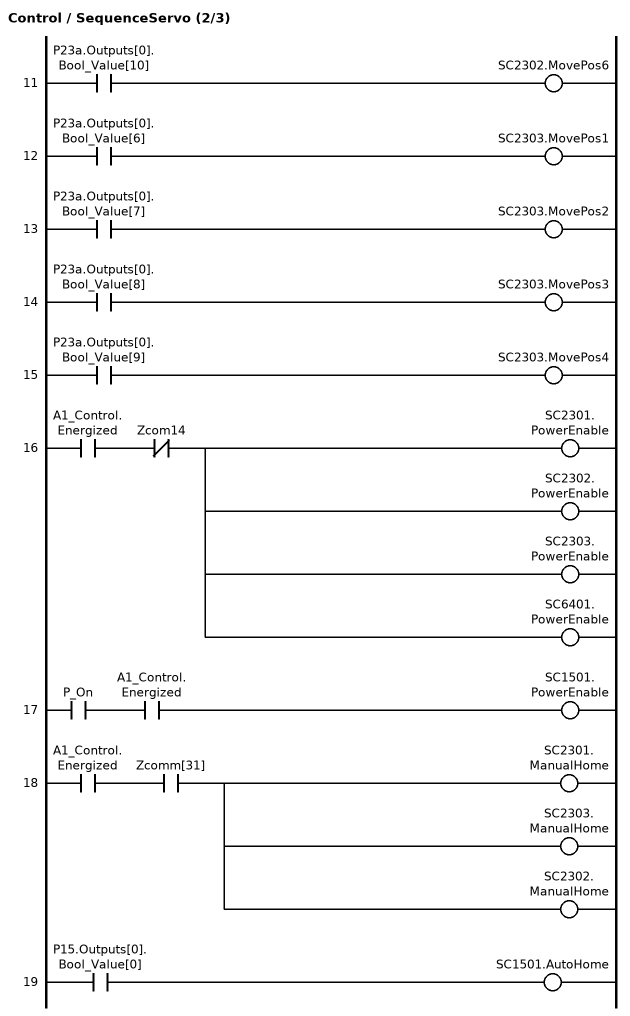
(* [picture p72: Control / SequenceServo, rungs 11-19] *)
(* Rung 11 *)
SC2302.MovePos6 := P23a.Outputs[0].Bool_Value[10];
(* Rung 12 *)
SC2303.MovePos1 := P23a.Outputs[0].Bool_Value[6];
(* Rung 13 *)
SC2303.MovePos2 := P23a.Outputs[0].Bool_Value[7];
(* Rung 14 *)
SC2303.MovePos3 := P23a.Outputs[0].Bool_Value[8];
(* Rung 15 *)
SC2303.MovePos4 := P23a.Outputs[0].Bool_Value[9];
(* Rung 16 *)
SC2301.PowerEnable := A1_Control.Energized AND NOT Zcom14;
SC2302.PowerEnable := A1_Control.Energized AND NOT Zcom14;
SC2303.PowerEnable := A1_Control.Energized AND NOT Zcom14;
SC6401.PowerEnable := A1_Control.Energized AND NOT Zcom14;
(* Rung 17 *)
SC1501.PowerEnable := P_On AND A1_Control.Energized;
(* Rung 18 *)
SC2301.ManualHome := A1_Control.Energized AND Zcomm[31];
SC2303.ManualHome := A1_Control.Energized AND Zcomm[31];
SC2302.ManualHome := A1_Control.Energized AND Zcomm[31];
(* Rung 19 *)
SC1501.AutoHome := P15.Outputs[0].Bool_Value[0];

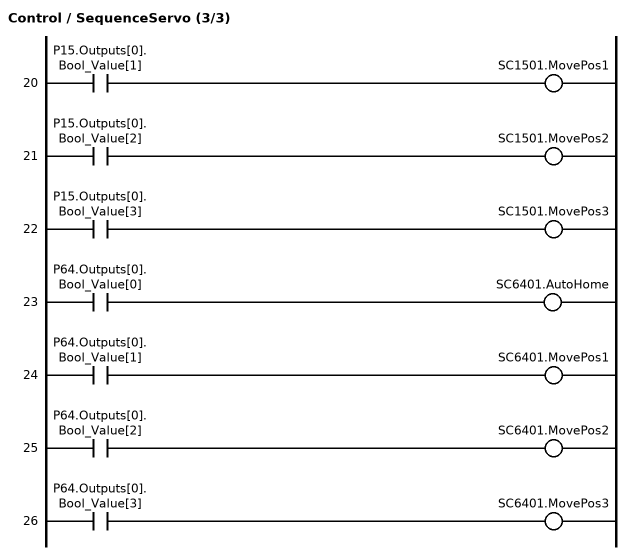
(* Rung 20 *)
SC1501.MovePos1 := P15.Outputs[0].Bool_Value[1];
(* Rung 21 *)
SC1501.MovePos2 := P15.Outputs[0].Bool_Value[2];
(* Rung 22 *)
SC1501.MovePos3 := P15.Outputs[0].Bool_Value[3];
(* Rung 23 *)
SC6401.AutoHome := P64.Outputs[0].Bool_Value[0];
(* Rung 24 *)
SC6401.MovePos1 := P64.Outputs[0].Bool_Value[1];
(* Rung 25 *)
SC6401.MovePos2 := P64.Outputs[0].Bool_Value[2];
(* Rung 26 *)
SC6401.MovePos3 := P64.Outputs[0].Bool_Value[3];

(* Section SequenceMotor: ladder, written here as Structured Text *)

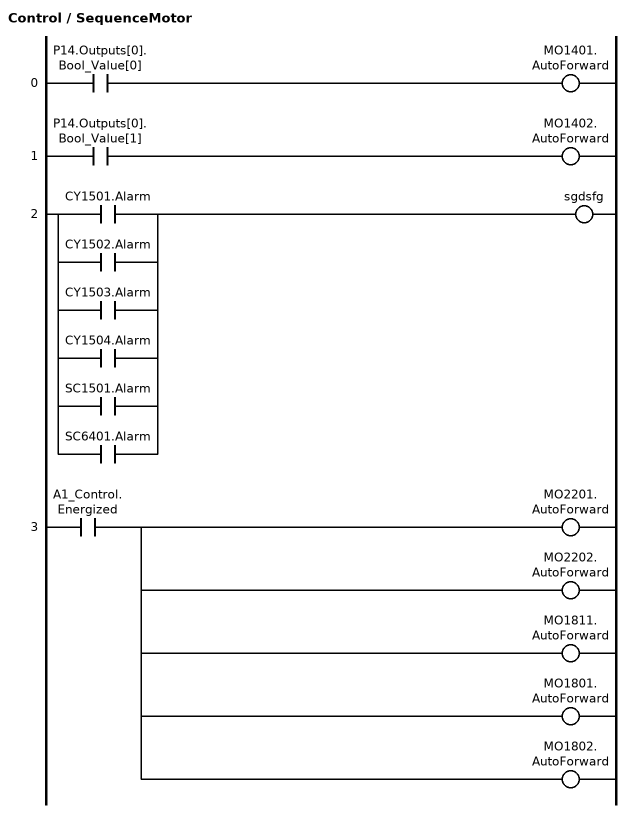
(* Rung 0 *)
MO1401.AutoForward := P14.Outputs[0].Bool_Value[0];
(* Rung 1 *)
MO1402.AutoForward := P14.Outputs[0].Bool_Value[1];
(* Rung 2 *)
sgdsfg := CY1501.Alarm OR CY1502.Alarm OR CY1503.Alarm OR CY1504.Alarm OR SC1501.Alarm OR SC6401.Alarm;
(* Rung 3 *)
MO2201.AutoForward := A1_Control.Energized;
MO2202.AutoForward := A1_Control.Energized;
MO1811.AutoForward := A1_Control.Energized;
MO1801.AutoForward := A1_Control.Energized;
MO1802.AutoForward := A1_Control.Energized;
END_PROGRAM

PROGRAM Outputs
VAR
    zcom : ARRAY[0..19] OF BOOL;
    IL0301_FB : MISCOUT;
    IL0302_FB : MISCOUT;
    IL0303_FB : MISCOUT;
    DO3501_FB : MISCOUT;
    DO1701_FB : MISCOUT;
    K1301_FB : MISCOUT;
    servo_drive_Error : BOOL;
    Actual_Value : DWORD;
    DO0351_FB : MISCOUT;
    CY1508_FB : CYL;
    CY1807_FB : CYL;
    CY1511_FB : CYL;
    CY1512_FB : CYL;
    CY3201_FB : CYL;
    CY3601_FB : CYL;
    SV1511_FB : MISCOUT;
    zcom1 : BOOL;
    zcom2 : BOOL;
    zcom6 : BOOL;
    CY4101_FB : CYL;
    CY4102_FB : CYL;
    CY4103_FB : CYL;
    CY4104_FB : CYL;
    CY4111_FB : CYL;
    CY4112_FB : CYL;
    CY4113_FB : CYL;
    CY4114_FB : CYL;
    CY4121_FB : CYL;
    CY4122_FB : CYL;
    CY4123_FB : CYL;
    CY4124_FB : CYL;
    Test2 : BOOL;
    SV : BOOL;
    SV4101_FB : MISCOUT;
    SV4102_FB : MISCOUT;
    SV4103_FB : MISCOUT;
    SV4104_FB : MISCOUT;
    XC0411_O1_15 : BOOL;
    MO1411_FB : MOTOR;
    zcom20 : BOOL;
    CY1401_FB : CYL;
    CY1402_FB : CYL;
    zcom21 : BOOL;
    zcom22 : BOOL;
    zcom23 : BOOL;
    zcom24 : BOOL;
    zcom_24 : BOOL;
    zcom_25 : BOOL;
    zcom_26 : BOOL;
    zcom_27 : BOOL;
    IL0304_FB : MiscOut;
    IL0305_FB : MiscOut;
    IL0306_FB : MiscOut;
    SV2701_FB : MiscOut;
    SV2702_FB : MiscOut;
    SV1501_FB : MiscOut;
    SV4111_FB : MiscOut;
    SV4112_FB : MiscOut;
    SV4113_FB : MiscOut;
    SV4114_FB : MiscOut;
    SV4121_FB : MiscOut;
    SV4122_FB : MiscOut;
    SV4123_FB : MiscOut;
    SV4124_FB : MiscOut;
    CY1501_FB : CYL;
    CY1502_FB : CYL;
    CY1503_FB : CYL;
    CY1504_FB : CYL;
    CY1505_FB : CYL;
    CY1506_FB : CYL;
    CY1507_FB : CYL;
    CY1801_FB : CYL;
    CY1802_FB : CYL;
    CY1804_FB : CYL;
    CY1803_FB : CYL;
    CY1805FB : CYL;
    CY1805_FB : CYL;
    CY1806_FB : CYL;
    CY2701_FB : CYL;
    CY3105_FB : CYL;
    SC1701_FB : Servo;
    SC2701_FB : Servo;
    SC_3201_FB : Servo;
    SC3201_FB : Servo;
    SC1702_FB : Servo;
    SC3601_FB : Servo;
    SC201_FB : Servo;
    SC3202_FB : Servo;
    MO2301_FB : Motor;
    MO3101_FB : MotorVSD;
    MO1401_FB : Motor;
    CY3102_FB : CYL;
    CY3103_FB : CYL;
    SC1701_Gear_SC1702 : MC_GearIn;
    A : BOOL;
    Vision_Test : Vision;
    Test4 : BOOL;
    Comm_DN : BOOL;
    SC1701_Gear_SC1702_Stop : MC_GearOut;
    GearStopMode : _eMC_OUT_MODE;
    CA2701_FB : Vision;
    CA1701_FB : Vision;
    SC1501_FB : Servo;
    CY1513_FB : CYL;
    CY1514_FB : CYL;
    CY1514_Extend : BOOL;
    CY1514_Retract : BOOL;
    CY3101_FB : CYL;
    SV4105_FB : MiscOut;
    SV4106_FB : MiscOut;
    SV4107_FB : MiscOut;
    SV4108_FB : MiscOut;
    SV4115_FB : MiscOut;
    SV4116_FB : MiscOut;
    SV4117_FB : MiscOut;
    SV4118_FB : MiscOut;
    SV4125_FB : MiscOut;
    SV4126_FB : MiscOut;
    SV4127_FB : MiscOut;
    SV4128_FB : MiscOut;
    CY1601_FB : CYL;
    CY1602_FB : CYL;
    CY2201_FB : CYL;
    CY2301_FB : CYL;
    CY2302_FB : CYL;
    CY2303_FB : CYL;
    CY2311_FB : CYL;
    CY2312_FB : CYL;
    CY2313_FB : CYL;
    CY2314_FB : CYL;
    CY2315_FB : CYL;
    CY2316_FB : CYL;
    CY2317_FB : CYL;
    CY2318_FB : CYL;
    CY2319_FB : CYL;
    CY2401_FB : CYL;
    CY2402_FB : CYL;
    MO1402_FB : Motor;
    MO3401_FB : MotorVSD;
    MO2311_FB : Motor;
    MO2201_FB : Motor;
    MO2202_FB : Motor;
    CY2501_A_FB : CYL;
    CY2501_B_FB : CYL;
    CY2501_C_FB : CYL;
    CY2501_D_FB : CYL;
    CY2502_A_FB : CYL;
    CY2502_B_FB : CYL;
    CY2503_A_FB : CYL;
    CY2503_B_FB : CYL;
    DO0301_FB : MiscOut;
    K0320_FB : MiscOut;
    K0321_FB : MiscOut;
    K0322_FB : MiscOut;
    K0323_FB : MiscOut;
    K4001_FB : MiscOut;
    DO3301_FB : MiscOut;
    DO3302_FB : MiscOut;
    SV0401_FB : MiscOut;
    SV2301_FB : MiscOut;
    SV2311_FB : MiscOut;
    SV2501_FB : MiscOut;
    SV2502_FB : MiscOut;
    CY3101_B_FB : CYL;
    CY3104_FB : CYL;
    CY3106_FB : CYL;
    CY2304_FB : CYL;
    CY2305_FB : CYL;
    CY2306_FB : CYL;
    CY2307_FB : CYL;
    CY2308_FB : CYL;
    CY2309_FB : CYL;
    M03401_FB : Motor;
    c : DINT;
    CY2501_FB : CYL;
    CY2502_FB : CYL;
    xc : BOOL;
    CY2201EX : BOOL;
    CY2201RT : BOOL;
    DO3502_FB : MiscOut;
    SV1502_FB : MiscOut;
    SV1503_FB : MiscOut;
    SV2511_FB : MiscOut;
    SV2512_FB : MiscOut;
    SV2521_FB : MiscOut;
    SV7101_FB : MiscOut;
    DO0320_FB : MiscOut;
    DO0350_FB : MiscOut;
    CY1811_FB : CYL;
    CY1812_FB : CYL;
    CY1701_FB : CYL;
    CY1702_FB : CYL;
    CY1703_FB : CYL;
    CY2521_FB : CYL;
    CY7101_FB : CYL;
    CY7102_FB : CYL;
    CY3401_FB : CYL;
    MO1801_FB : Motor;
    MO1811_FB : Motor;
    MO1701_FB : Motor;
    SC6401_FB : Servo;
    SC2301_FB : Servo;
    SC2302_FB : Servo;
    SC2303_FB : Servo;
    DO3511_FB : MiscOut;
    CY3402_FB : CYL;
    M03101_FB : Motor;
    MO2701_FB : Motor;
    MO2702_FB : Motor;
    MO1802_FB : Motor;
    SV2522_FB : MiscOut;
END_VAR
VAR_EXTERNAL
    CY1601 : CylinderD;
    A1_Control : System;
    CY2502 : CylinderD;
    CY2501 : CylinderD;
    CY2402 : CylinderD;
    CY2401 : CylinderD;
    CY2302 : CylinderD;
    CY2303 : CylinderD;
    CY2301 : CylinderD;
    SC2701 : ServoD;
    MO1402 : MotorD;
    MO2301 : MotorD;
    MO2201 : MotorD;
    MO2202 : MotorD;
    IL0302 : MiscOutD;
    IL0303 : MiscOutD;
    DO0301 : MiscOutD;
    DO3301 : MiscOutD;
    DO3302 : MiscOutD;
    SV0401 : MiscOutD;
    SV1501 : MiscOutD;
    SV2301 : MiscOutD;
    SV2501 : MiscOutD;
    SV2502 : MiscOutD;
    IL0301 : MiscOutD;
    CY2304 : CylinderD;
    RO4001_I_PalletizingDone : BOOL;
    PS2501 : MiscInD;
    P27 : SequenceD;
    SKU_Select : DINT;
    DO3502 : MiscOutD;
    DO3501 : MiscOutD;
    K1301 : MiscOutD;
    SV2701 : MiscOutD;
    SV1502 : MiscOutD;
    SV1503 : MiscOutD;
    SV2511 : MiscOutD;
    SV2512 : MiscOutD;
    SV2521 : MiscOutD;
    SV7101 : MiscOutD;
    DO320 : MiscOutD;
    DO0320 : MiscOutD;
    DO0350 : MiscOutD;
    CY1502 : CylinderD;
    CY1503 : CylinderD;
    CY1504 : CylinderD;
    CY1811 : CylinderD;
    CY1701 : CylinderD;
    CY1702 : CylinderD;
    CY1703 : CylinderD;
    CY2521 : CylinderD;
    CY7101 : CylinderD;
    CY7102 : CylinderD;
    CY3401 : CylinderD;
    CY3402 : CylinderD;
    MO1801 : MotorD;
    MO1811 : MotorD;
    MO1701 : MotorD;
    MO3101 : MotorD;
    SC1501 : ServoD;
    SC1501_Ax : _sAXIS_REF;
    SC6401 : ServoD;
    SC6401_Ax : _sAXIS_REF;
    SC2301 : ServoD;
    SC2301_Ax : _sAXIS_REF;
    SC2302 : ServoD;
    SC2302_Ax : _sAXIS_REF;
    SC2303 : ServoD;
    SC2303_Ax : _sAXIS_REF;
    XC0301_6_I : ARRAY[0..15] OF BOOL;
    XC0301_7_I : ARRAY[0..15] OF BOOL;
    XC0301_8_O : ARRAY[0..15] OF BOol;
    IL0304 : MiscOutD;
    XC0301_9_O : ARRAY[0..15] OF BOOL;
    XC0320_1_O_2 : BOOL;
    XC0320_1_O_3 : BOOL;
    XC0320_1_O_4 : BOOL;
    XC0320_1_I_5 : BOOL;
    XC0320_1_I_6 : BOOL;
    XC0320_1_I_7 : BOOL;
    XC0320_1_I_8 : BOOL;
    XC0320_1_I_9 : BOOL;
    XC0320_1_I_10 : BOOL;
    XC0320_2_O_0 : BOOL;
    XC0320_2_O_1 : BOOL;
    XC0320_2_O_2 : BOOL;
    XC0320_2_O_3 : BOOL;
    XC0320_2_O_4 : BOOL;
    XC0320_2_O_5 : BOOL;
    DO3511 : MiscOutD;
    XC0320_2_O_6 : BOOL;
    XC0320_3_O_0 : BOOL;
    XC0320_3_O_1 : BOOL;
    XC0320_3_O_2 : BOOL;
    XC0320_3_O_3 : BOOL;
    XC0320_3_I_4 : BOOL;
    XC0320_3_I_5 : BOOL;
    XC0320_3_I_6 : BOOL;
    XC0320_3_I_7 : BOOL;
    XC0320_3_I_8 : BOOL;
    XC0320_3_I_9 : BOOL;
    XC0320_4_I_0 : BOOL;
    XC0320_4_I_1 : BOOL;
    XC0320_4_I_2 : BOOL;
    XC0320_4_I_3 : BOOL;
    XC0320_4_I_4 : BOOL;
    XC0320_4_I_5 : BOOL;
    XC0320_4_I_6 : BOOL;
    XC0320_4_I_7 : BOOL;
    XC0320_4_I_8 : BOOL;
    XC0320_4_I_9 : BOOL;
    XC0320_4_I_10 : BOOL;
    XC0320_4_I_11 : BOOL;
    XC0320_4_I_12 : BOOL;
    XC0320_4_I_13 : BOOL;
    XC0320_4_I_14 : BOOL;
    XC0320_4_I_15 : BOOL;
    XC0320_5_I_0 : BOOL;
    XC0320_5_I_1 : BOOL;
    XC0320_5_I_2 : BOOL;
    XC0320_5_I_3 : BOOL;
    MO1401 : MotorD;
    MO3401 : MotorD;
    CY1501 : CylinderD;
    Ketan : WORD;
    Sandesh : WORD;
    jhsac : BOOL;
    CY2305 : CylinderD;
    XC0320_1_I_0 : BOOL;
    XC0320_1_I_1 : BOOL;
    XC0320_1_I_11 : BOOL;
    XC0320_1_I_12 : BOOL;
    XC0320_3_I_14 : BOOL;
    XC0320_3_I_15 : BOOL;
    XC0320_5_O_8 : BOOL;
    XC0320_5_O_9 : BOOL;
    XC0320_5_O_10 : BOOL;
    MO2701 : MotorD;
    MO2702 : MotorD;
    MO1802 : MotorD;
    SV2522 : MiscOutD;
    A0XC0401_1_I_4 : BOOL;
    A0XC0401_1_I_5 : BOOL;
    A0XC0401_1_I_6 : BOOL;
    A0XC0401_1_I_7 : BOOL;
    CY2701 : CylinderD;
    A0XC0401_1_I_11 : BOOL;
    A0XC0401_1_I_12 : BOOL;
    A0XC0401_1_O_0 : BOOL;
    A0XC0401_1_O_1 : BOOL;
    A0XC0401_1_O_3 : BOOL;
    A0XC0401_1_O_4 : BOOL;
    A0XC0401_1_O_5 : BOOL;
    A0XC0401_1_O_2 : BOOL;
    A0XC0401_2_O_0 : BOOL;
    A0XC0401_2_O_1 : BOOL;
    A0XC0401_1_O_6 : BOOL;
    A0XC0401_1_O_7 : BOOL;
    XC0320_1_I_15 : BOOL;
    XC0320_1_I_14 : BOOL;
    A0XC0401_2_O_2 : BOOL;
    A0XC0401_2_O_3 : BOOL;
    A0XC0401_2_O_4 : BOOL;
    A0XC0401_2_O_5 : BOOL;
    A0XC0401_2_O_6 : BOOL;
    A0XC0401_2_O_7 : BOOL;
END_VAR
VAR_EXTERNAL CONSTANT
    SC1501Ax : _sAXIS_REF;
    SC2301Ax : _sAXIS_REF;
    SC2302Ax : _sAXIS_REF;
    SC2303Ax : _sAXIS_REF;
    SC6401Ax : _sAXIS_REF;
END_VAR
VAR_EXTERNAL
    XC0320_2_O_8 : BOOL;
    XC0320_2_O_9 : BOOL;
    A0XC0401_3_O_0 : BOOL;
    A0XC0401_3_O_1 : BOOL;
    A0XC0401_3_O_2 : BOOL;
    A0XC0401_3_O_3 : BOOL;
    A0XC0401_3_O_4 : BOOL;
    A0XC0401_3_O_5 : BOOL;
    A0XC0401_3_O_6 : BOOL;
    A0XC0401_3_O_7 : BOOL;
    XC0320_2_I_0 : BOOL;
    XC0320_2_I_1 : BOOL;
END_VAR

(* Section IDMiscOut: ladder, written here as Structured Text *)

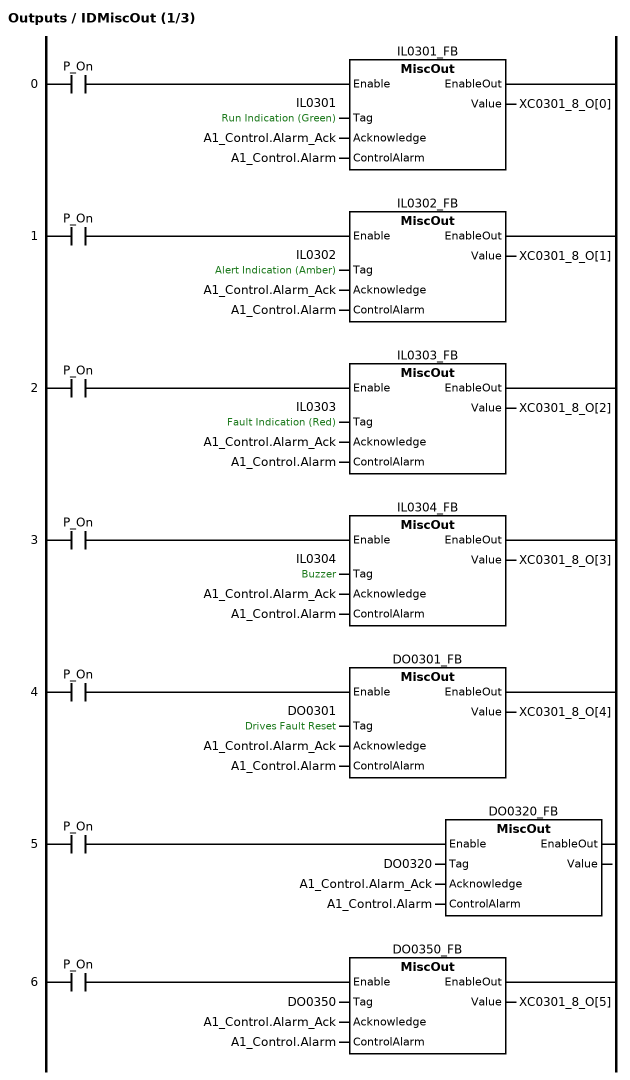
(* Rung 0 *)
IL0301_FB(Enable := P_On, Tag := IL0301, Acknowledge := A1_Control.Alarm_Ack, ControlAlarm := A1_Control.Alarm, Value => XC0301_8_O[0]);
(* Rung 1 *)
IL0302_FB(Enable := P_On, Tag := IL0302, Acknowledge := A1_Control.Alarm_Ack, ControlAlarm := A1_Control.Alarm, Value => XC0301_8_O[1]);
(* Rung 2 *)
IL0303_FB(Enable := P_On, Tag := IL0303, Acknowledge := A1_Control.Alarm_Ack, ControlAlarm := A1_Control.Alarm, Value => XC0301_8_O[2]);
(* Rung 3 *)
IL0304_FB(Enable := P_On, Tag := IL0304, Acknowledge := A1_Control.Alarm_Ack, ControlAlarm := A1_Control.Alarm, Value => XC0301_8_O[3]);
(* Rung 4 *)
DO0301_FB(Enable := P_On, Tag := DO0301, Acknowledge := A1_Control.Alarm_Ack, ControlAlarm := A1_Control.Alarm, Value => XC0301_8_O[4]);
(* Rung 5 *)
DO0320_FB(Enable := P_On, Tag := DO0320, Acknowledge := A1_Control.Alarm_Ack, ControlAlarm := A1_Control.Alarm);
(* notes on elements: Safety Reset *)
(* Rung 6 *)
DO0350_FB(Enable := P_On, Tag := DO0350, Acknowledge := A1_Control.Alarm_Ack, ControlAlarm := A1_Control.Alarm, Value => XC0301_8_O[5]);
(* notes on elements: Upstream Signal *)

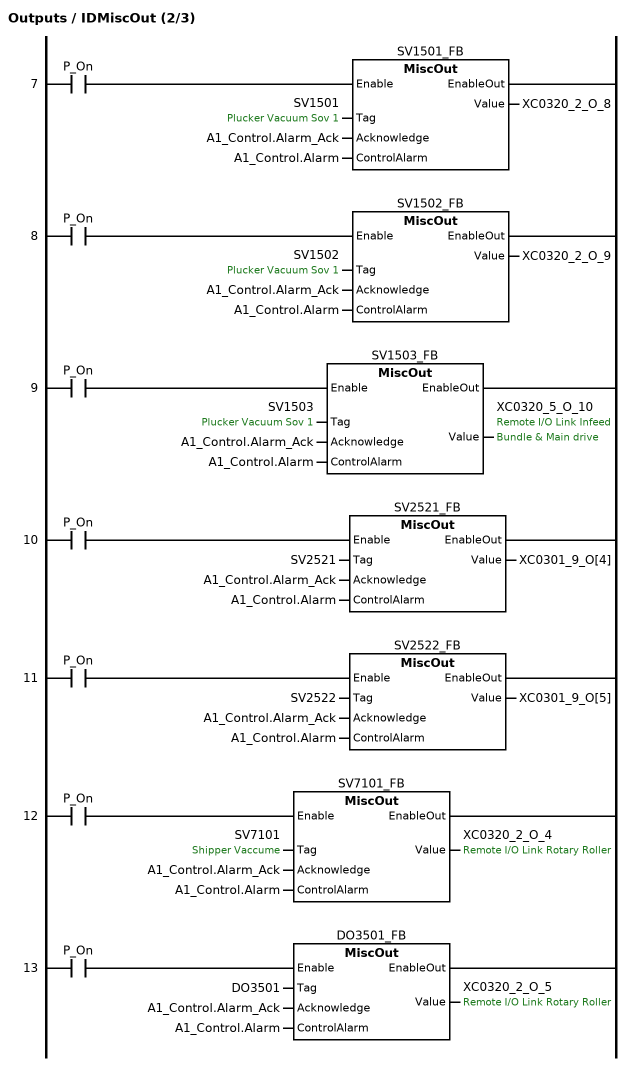
(* Rung 7 *)
SV1501_FB(Enable := P_On, Tag := SV1501, Acknowledge := A1_Control.Alarm_Ack, ControlAlarm := A1_Control.Alarm, Value => XC0320_2_O_8);
(* notes on elements: Plucker Vacuum Sov 1 *)
(* Rung 8 *)
SV1502_FB(Enable := P_On, Tag := SV1502, Acknowledge := A1_Control.Alarm_Ack, ControlAlarm := A1_Control.Alarm, Value => XC0320_2_O_9);
(* notes on elements: Plucker Vacuum Sov 2 *)
(* Rung 9 *)
SV1503_FB(Enable := P_On, Tag := SV1503, Acknowledge := A1_Control.Alarm_Ack, ControlAlarm := A1_Control.Alarm, Value => XC0320_5_O_10);
(* notes on elements: Plucker Vacuum Sov 3 *)
(* Rung 10 *)
SV2521_FB(Enable := P_On, Tag := SV2521, Acknowledge := A1_Control.Alarm_Ack, ControlAlarm := A1_Control.Alarm, Value => XC0301_9_O[4]);
(* notes on elements: Vacuum Solenoid *)
(* Rung 11 *)
SV2522_FB(Enable := P_On, Tag := SV2522, Acknowledge := A1_Control.Alarm_Ack, ControlAlarm := A1_Control.Alarm, Value => XC0301_9_O[5]);
(* notes on elements: layerboard pickhead purging *)
(* Rung 12 *)
SV7101_FB(Enable := P_On, Tag := SV7101, Acknowledge := A1_Control.Alarm_Ack, ControlAlarm := A1_Control.Alarm, Value => XC0320_2_O_4);
(* notes on elements: Shipper Vacuum *)
(* Rung 13 *)
DO3501_FB(Enable := P_On, Tag := DO3501, Acknowledge := A1_Control.Alarm_Ack, ControlAlarm := A1_Control.Alarm, Value => XC0320_2_O_5);
(* notes on elements: Pre-Label Applicator Trigger Signal *)

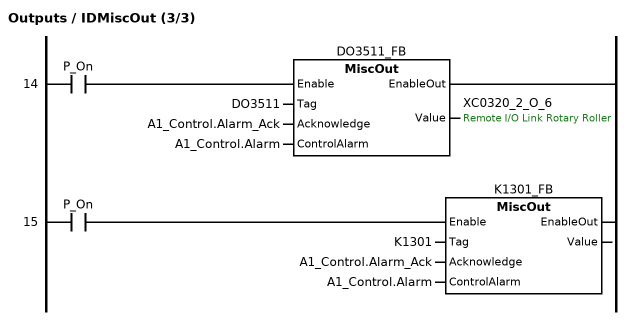
(* Rung 14 *)
DO3511_FB(Enable := P_On, Tag := DO3511, Acknowledge := A1_Control.Alarm_Ack, ControlAlarm := A1_Control.Alarm, Value => XC0320_2_O_6);
(* notes on elements: OCR Camera Trigger Signal *)
(* Rung 15 *)
K1301_FB(Enable := P_On, Tag := K1301, Acknowledge := A1_Control.Alarm_Ack, ControlAlarm := A1_Control.Alarm);
(* notes on elements: Guard Door Coil Supply *)

(* Section IDCylinder: ladder, written here as Structured Text *)

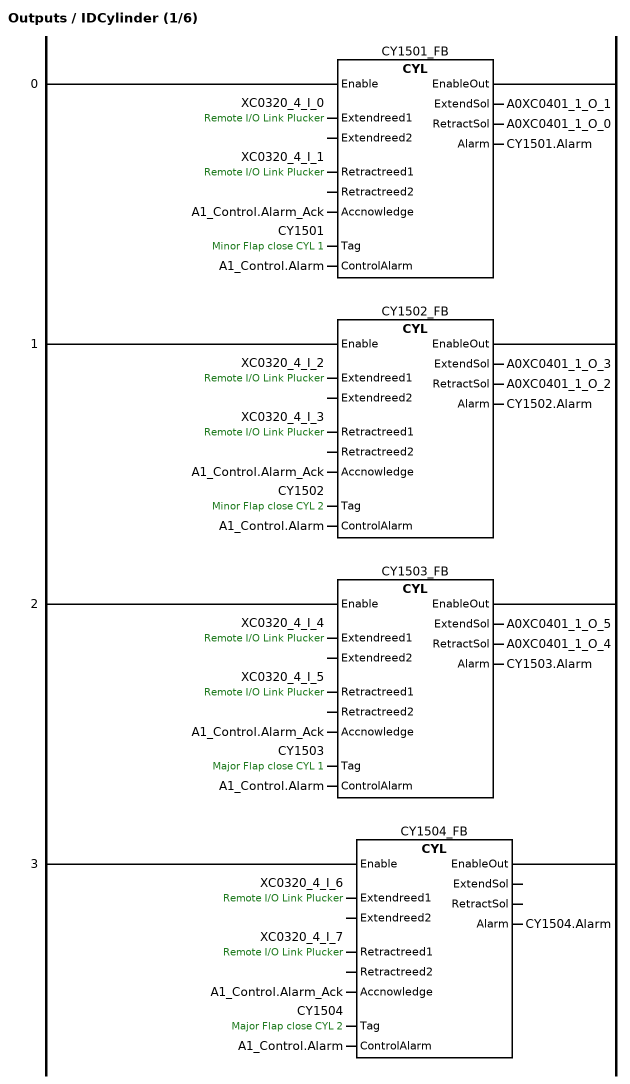
(* Rung 0 *)
CY1501_FB(Enable := TRUE, Extendreed1 := XC0320_4_I_0, Retractreed1 := XC0320_4_I_1, Accnowledge := A1_Control.Alarm_Ack, Tag := CY1501, ControlAlarm := A1_Control.Alarm, ExtendSol => A0XC0401_1_O_1, RetractSol => A0XC0401_1_O_0, Alarm => CY1501.Alarm);
(* notes on elements: Minor Flap close CYL 1 *)
(* Rung 1 *)
CY1502_FB(Enable := TRUE, Extendreed1 := XC0320_4_I_2, Retractreed1 := XC0320_4_I_3, Accnowledge := A1_Control.Alarm_Ack, Tag := CY1502, ControlAlarm := A1_Control.Alarm, ExtendSol => A0XC0401_1_O_3, RetractSol => A0XC0401_1_O_2, Alarm => CY1502.Alarm);
(* notes on elements: Minor Flap close CYL 2 *)
(* Rung 2 *)
CY1503_FB(Enable := TRUE, Extendreed1 := XC0320_4_I_4, Retractreed1 := XC0320_4_I_5, Accnowledge := A1_Control.Alarm_Ack, Tag := CY1503, ControlAlarm := A1_Control.Alarm, ExtendSol => A0XC0401_1_O_5, RetractSol => A0XC0401_1_O_4, Alarm => CY1503.Alarm);
(* notes on elements: Major Flap close CYL 1 *)
(* Rung 3 *)
CY1504_FB(Enable := TRUE, Extendreed1 := XC0320_4_I_6, Retractreed1 := XC0320_4_I_7, Accnowledge := A1_Control.Alarm_Ack, Tag := CY1504, ControlAlarm := A1_Control.Alarm, Alarm => CY1504.Alarm);
(* notes on elements: Major Flap close CYL 2 *)

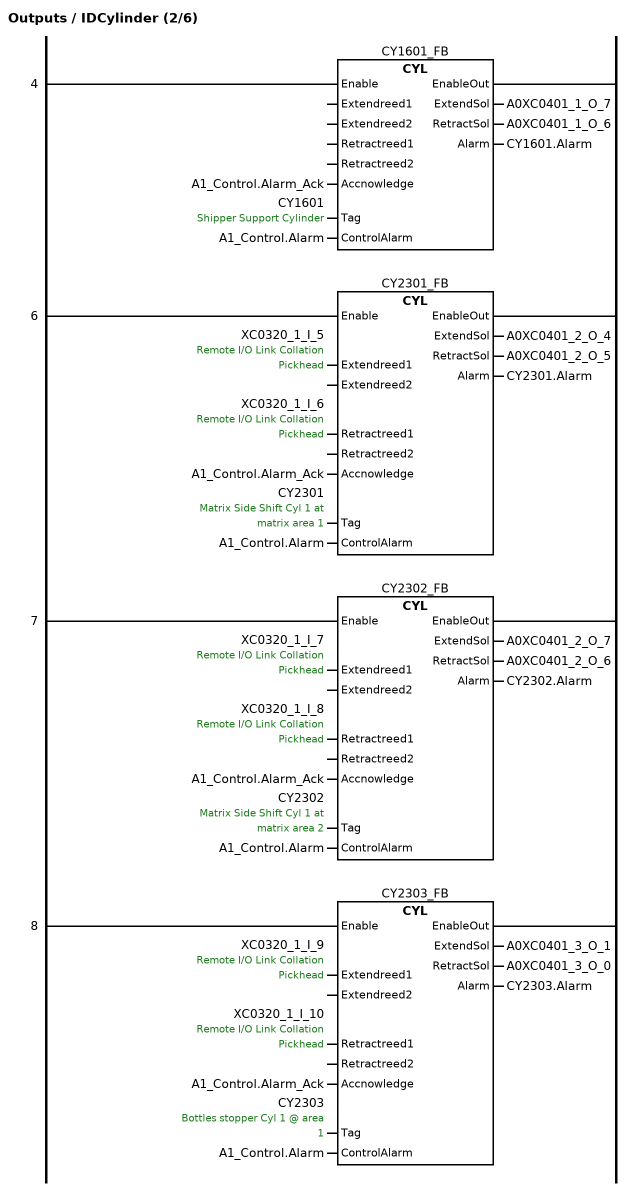
(* Rung 4 *)
CY1601_FB(Enable := TRUE, Accnowledge := A1_Control.Alarm_Ack, Tag := CY1601, ControlAlarm := A1_Control.Alarm, ExtendSol => A0XC0401_1_O_7, RetractSol => A0XC0401_1_O_6, Alarm => CY1601.Alarm);
(* Rung 6 *)
CY2301_FB(Enable := TRUE, Extendreed1 := XC0320_1_I_5, Retractreed1 := XC0320_1_I_6, Accnowledge := A1_Control.Alarm_Ack, Tag := CY2301, ControlAlarm := A1_Control.Alarm, ExtendSol => A0XC0401_2_O_4, RetractSol => A0XC0401_2_O_5, Alarm => CY2301.Alarm);
(* notes on elements: Matrix Side Shift Cyl 1 at matrix area 1 *)
(* Rung 7 *)
CY2302_FB(Enable := TRUE, Extendreed1 := XC0320_1_I_7, Retractreed1 := XC0320_1_I_8, Accnowledge := A1_Control.Alarm_Ack, Tag := CY2302, ControlAlarm := A1_Control.Alarm, ExtendSol => A0XC0401_2_O_7, RetractSol => A0XC0401_2_O_6, Alarm => CY2302.Alarm);
(* notes on elements: Matrix Side Shift Cyl 2 at matrix area 2 *)
(* Rung 8 *)
CY2303_FB(Enable := TRUE, Extendreed1 := XC0320_1_I_9, Retractreed1 := XC0320_1_I_10, Accnowledge := A1_Control.Alarm_Ack, Tag := CY2303, ControlAlarm := A1_Control.Alarm, ExtendSol => A0XC0401_3_O_1, RetractSol => A0XC0401_3_O_0, Alarm => CY2303.Alarm);

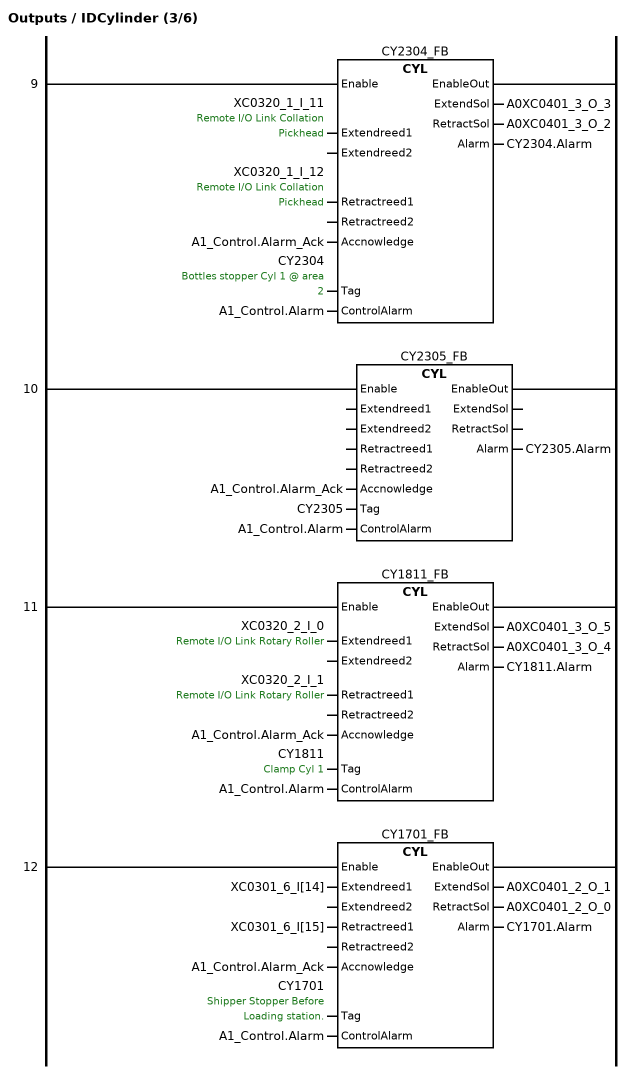
(* Rung 9 *)
CY2304_FB(Enable := TRUE, Extendreed1 := XC0320_1_I_11, Retractreed1 := XC0320_1_I_12, Accnowledge := A1_Control.Alarm_Ack, Tag := CY2304, ControlAlarm := A1_Control.Alarm, ExtendSol => A0XC0401_3_O_3, RetractSol => A0XC0401_3_O_2, Alarm => CY2304.Alarm);
(* notes on elements: Bottles stopper Cyl 1 @ area 1 *)
(* Rung 10 *)
CY2305_FB(Enable := TRUE, Accnowledge := A1_Control.Alarm_Ack, Tag := CY2305, ControlAlarm := A1_Control.Alarm, Alarm => CY2305.Alarm);
(* notes on elements: Bottles stopper Cyl 2 @ area 2 *)
(* Rung 11 *)
CY1811_FB(Enable := TRUE, Extendreed1 := XC0320_2_I_0, Retractreed1 := XC0320_2_I_1, Accnowledge := A1_Control.Alarm_Ack, Tag := CY1811, ControlAlarm := A1_Control.Alarm, ExtendSol => A0XC0401_3_O_5, RetractSol => A0XC0401_3_O_4, Alarm => CY1811.Alarm);
(* notes on elements: Clamp Cyl 1 *)
(* Rung 12 *)
CY1701_FB(Enable := TRUE, Extendreed1 := XC0301_6_I[14], Retractreed1 := XC0301_6_I[15], Accnowledge := A1_Control.Alarm_Ack, Tag := CY1701, ControlAlarm := A1_Control.Alarm, ExtendSol => A0XC0401_2_O_1, RetractSol => A0XC0401_2_O_0, Alarm => CY1701.Alarm);
(* notes on elements: Shipper Stopper Before Loading station. *)

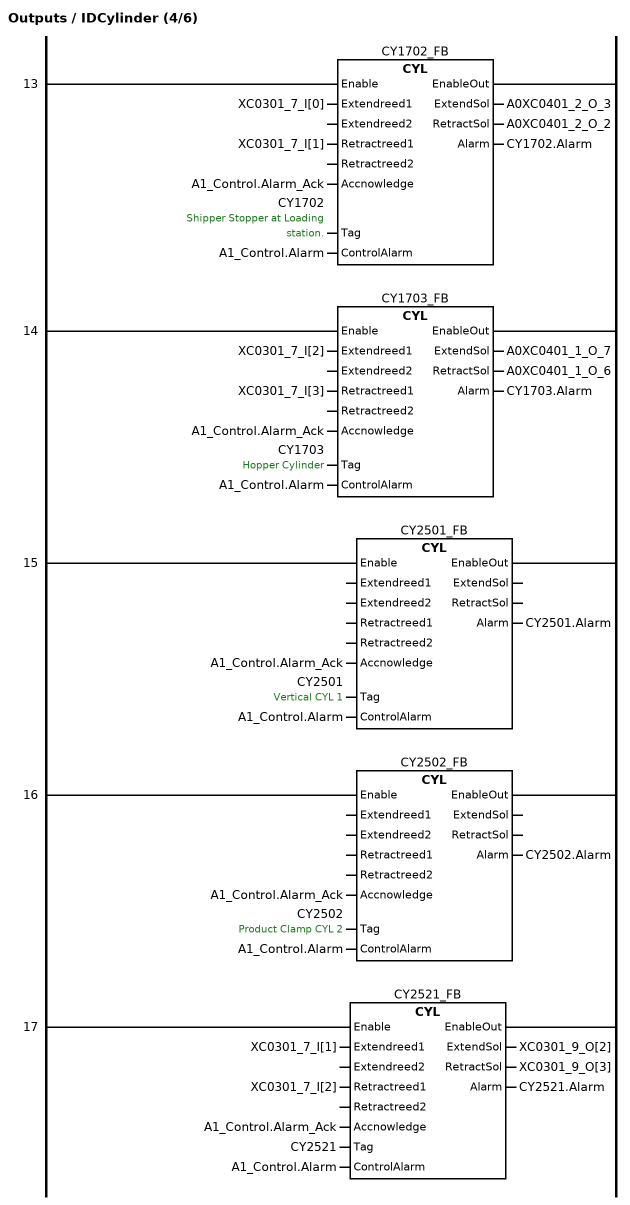
(* Rung 13 *)
CY1702_FB(Enable := TRUE, Extendreed1 := XC0301_7_I[0], Retractreed1 := XC0301_7_I[1], Accnowledge := A1_Control.Alarm_Ack, Tag := CY1702, ControlAlarm := A1_Control.Alarm, ExtendSol => A0XC0401_2_O_3, RetractSol => A0XC0401_2_O_2, Alarm => CY1702.Alarm);
(* notes on elements: Shipper Stopper at Loading station. *)
(* Rung 14 *)
CY1703_FB(Enable := TRUE, Extendreed1 := XC0301_7_I[2], Retractreed1 := XC0301_7_I[3], Accnowledge := A1_Control.Alarm_Ack, Tag := CY1703, ControlAlarm := A1_Control.Alarm, ExtendSol => A0XC0401_1_O_7, RetractSol => A0XC0401_1_O_6, Alarm => CY1703.Alarm);
(* notes on elements: Hopper Flap Open CYL *)
(* Rung 15 *)
CY2501_FB(Enable := TRUE, Accnowledge := A1_Control.Alarm_Ack, Tag := CY2501, ControlAlarm := A1_Control.Alarm, Alarm => CY2501.Alarm);
(* notes on elements: Bottle Clamp Cyl 1 *)
(* Rung 16 *)
CY2502_FB(Enable := TRUE, Accnowledge := A1_Control.Alarm_Ack, Tag := CY2502, ControlAlarm := A1_Control.Alarm, Alarm => CY2502.Alarm);
(* notes on elements: Bundle matrix clamp Cyl 1 *)
(* Rung 17 *)
CY2521_FB(Enable := TRUE, Extendreed1 := XC0301_7_I[1], Retractreed1 := XC0301_7_I[2], Accnowledge := A1_Control.Alarm_Ack, Tag := CY2521, ControlAlarm := A1_Control.Alarm, ExtendSol => XC0301_9_O[2], RetractSol => XC0301_9_O[3], Alarm => CY2521.Alarm);
(* notes on elements: Pickhead Rotary CYL *)

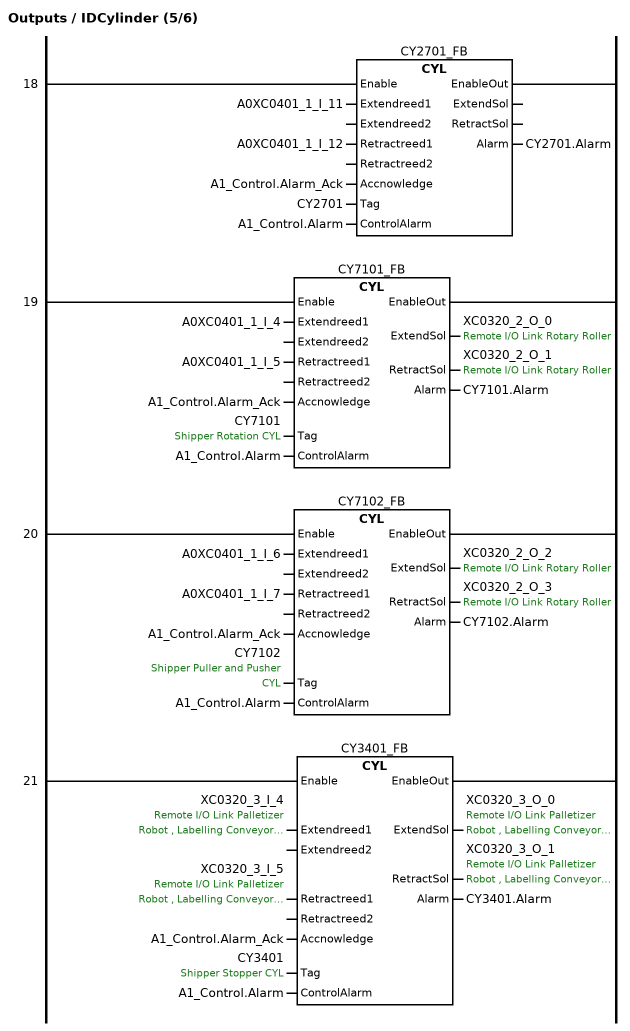
(* Rung 18 *)
CY2701_FB(Enable := TRUE, Extendreed1 := A0XC0401_1_I_11, Retractreed1 := A0XC0401_1_I_12, Accnowledge := A1_Control.Alarm_Ack, Tag := CY2701, ControlAlarm := A1_Control.Alarm, Alarm => CY2701.Alarm);
(* notes on elements: Minor Flap Close CYL @ Top Tapping *)
(* Rung 19 *)
CY7101_FB(Enable := TRUE, Extendreed1 := A0XC0401_1_I_4, Retractreed1 := A0XC0401_1_I_5, Accnowledge := A1_Control.Alarm_Ack, Tag := CY7101, ControlAlarm := A1_Control.Alarm, ExtendSol => XC0320_2_O_0, RetractSol => XC0320_2_O_1, Alarm => CY7101.Alarm);
(* notes on elements: Shipper Rotation CYL *)
(* Rung 20 *)
CY7102_FB(Enable := TRUE, Extendreed1 := A0XC0401_1_I_6, Retractreed1 := A0XC0401_1_I_7, Accnowledge := A1_Control.Alarm_Ack, Tag := CY7102, ControlAlarm := A1_Control.Alarm, ExtendSol => XC0320_2_O_2, RetractSol => XC0320_2_O_3, Alarm => CY7102.Alarm);
(* notes on elements: Shipper Puller and Pusher CYL *)
(* Rung 21 *)
CY3401_FB(Enable := TRUE, Extendreed1 := XC0320_3_I_4, Retractreed1 := XC0320_3_I_5, Accnowledge := A1_Control.Alarm_Ack, Tag := CY3401, ControlAlarm := A1_Control.Alarm, ExtendSol => XC0320_3_O_0, RetractSol => XC0320_3_O_1, Alarm => CY3401.Alarm);
(* notes on elements: Shipper Stopper Cylinder *)

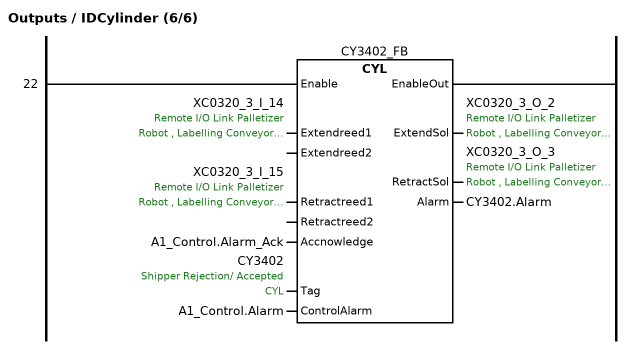
(* Rung 22 *)
CY3402_FB(Enable := TRUE, Extendreed1 := XC0320_3_I_14, Retractreed1 := XC0320_3_I_15, Accnowledge := A1_Control.Alarm_Ack, Tag := CY3402, ControlAlarm := A1_Control.Alarm, ExtendSol => XC0320_3_O_2, RetractSol => XC0320_3_O_3, Alarm => CY3402.Alarm);
(* notes on elements: Shipper Rejection CYL *)

(* Section IDServo: ladder, written here as Structured Text *)

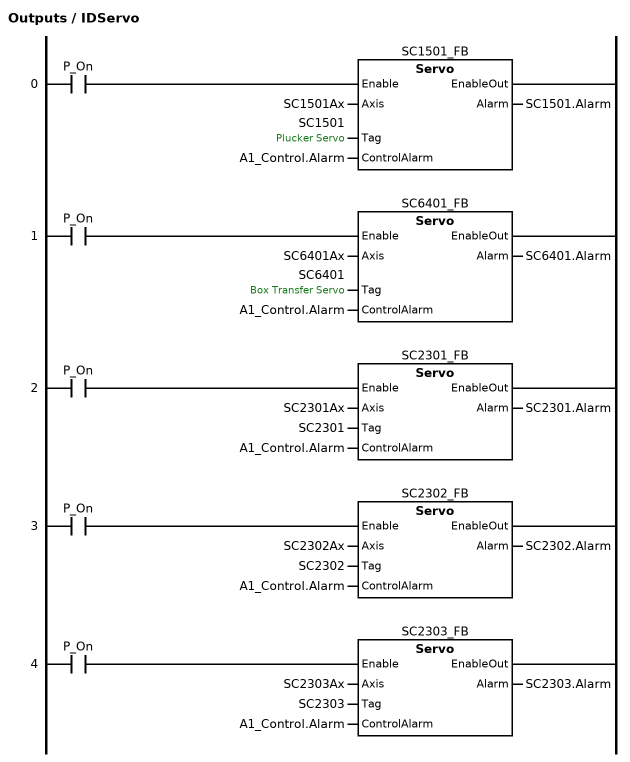
(* Rung 0 *)
SC1501_FB(Enable := P_On, Axis := SC1501Ax, Tag := SC1501, ControlAlarm := A1_Control.Alarm, Alarm => SC1501.Alarm);
(* notes on elements: Plucker Servo Motor *)
(* Rung 1 *)
SC6401_FB(Enable := P_On, Axis := SC6401Ax, Tag := SC6401, ControlAlarm := A1_Control.Alarm, Alarm => SC6401.Alarm);
(* notes on elements: Box Transfer Servo Motor *)
(* Rung 2 *)
SC2301_FB(Enable := P_On, Axis := SC2301Ax, Tag := SC2301, ControlAlarm := A1_Control.Alarm, Alarm => SC2301.Alarm);
(* notes on elements: Side Shift Servo Motor 1 *)
(* Rung 3 *)
SC2302_FB(Enable := P_On, Axis := SC2302Ax, Tag := SC2302, ControlAlarm := A1_Control.Alarm, Alarm => SC2302.Alarm);
(* notes on elements: Side Shift Servo Motor 2 *)
(* Rung 4 *)
SC2303_FB(Enable := P_On, Axis := SC2303Ax, Tag := SC2303, ControlAlarm := A1_Control.Alarm, Alarm => SC2303.Alarm);
(* notes on elements: Side Shift Servo Motor 3 *)

(* Section IDMotor: ladder, written here as Structured Text *)

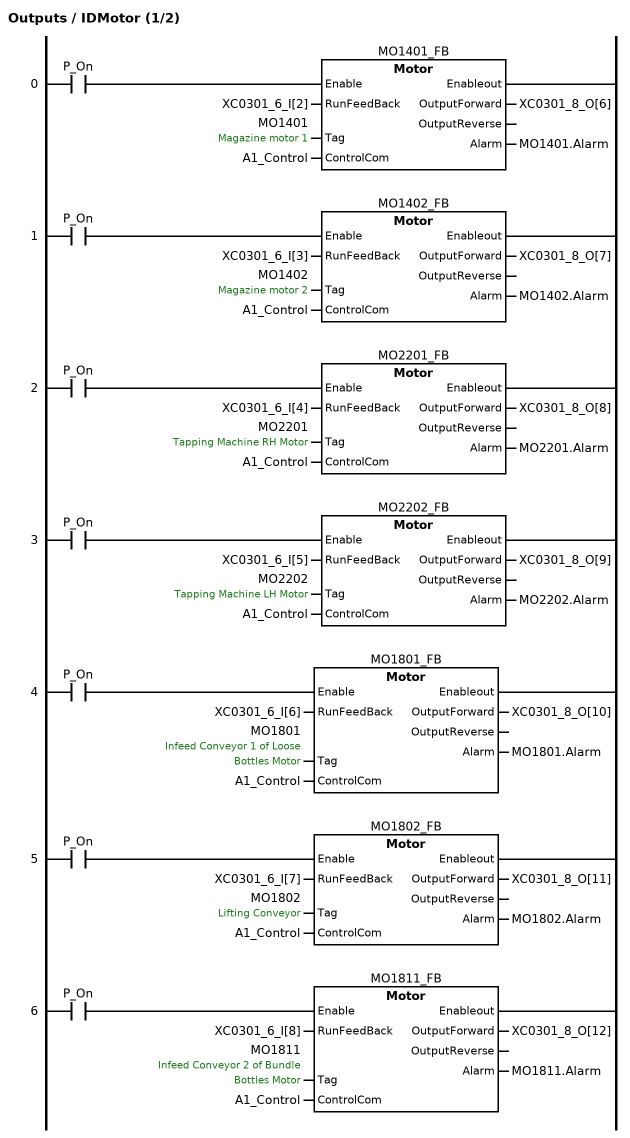
(* Rung 0 *)
MO1401_FB(Enable := P_On, RunFeedBack := XC0301_6_I[2], Tag := MO1401, ControlCom := A1_Control, OutputForward => XC0301_8_O[6], Alarm => MO1401.Alarm);
(* notes on elements: Magazine motor 1 *)
(* Rung 1 *)
MO1402_FB(Enable := P_On, RunFeedBack := XC0301_6_I[3], Tag := MO1402, ControlCom := A1_Control, OutputForward => XC0301_8_O[7], Alarm => MO1402.Alarm);
(* notes on elements: Magazine motor 2 *)
(* Rung 2 *)
MO2201_FB(Enable := P_On, RunFeedBack := XC0301_6_I[4], Tag := MO2201, ControlCom := A1_Control, OutputForward => XC0301_8_O[8], Alarm => MO2201.Alarm);
(* notes on elements: Bottom Taping RH Motor *)
(* Rung 3 *)
MO2202_FB(Enable := P_On, RunFeedBack := XC0301_6_I[5], Tag := MO2202, ControlCom := A1_Control, OutputForward => XC0301_8_O[9], Alarm => MO2202.Alarm);
(* notes on elements: Bottom Taping LH Motor *)
(* Rung 4 *)
MO1801_FB(Enable := P_On, RunFeedBack := XC0301_6_I[6], Tag := MO1801, ControlCom := A1_Control, OutputForward => XC0301_8_O[10], Alarm => MO1801.Alarm);
(* notes on elements: Infeed conveyor of Loose Bottle *)
(* Rung 5 *)
MO1802_FB(Enable := P_On, RunFeedBack := XC0301_6_I[7], Tag := MO1802, ControlCom := A1_Control, OutputForward => XC0301_8_O[11], Alarm => MO1802.Alarm);
(* notes on elements: Lifting Conveyor *)
(* Rung 6 *)
MO1811_FB(Enable := P_On, RunFeedBack := XC0301_6_I[8], Tag := MO1811, ControlCom := A1_Control, OutputForward => XC0301_8_O[12], Alarm => MO1811.Alarm);
(* notes on elements: Infeed Conveyor of Bundle Bottles *)

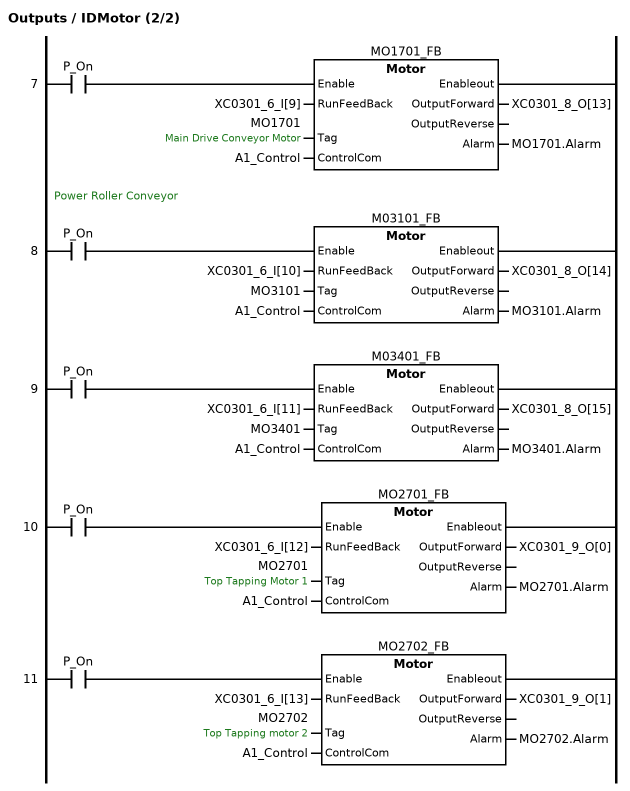
(* Rung 7 *)
MO1701_FB(Enable := P_On, RunFeedBack := XC0301_6_I[9], Tag := MO1701, ControlCom := A1_Control, OutputForward => XC0301_8_O[13], Alarm => MO1701.Alarm);
(* notes on elements: Main Drive Conveyor Motor *)
(* Rung 8: Power Roller Conveyor *)
M03101_FB(Enable := P_On, RunFeedBack := XC0301_6_I[10], Tag := MO3101, ControlCom := A1_Control, OutputForward => XC0301_8_O[14], Alarm => MO3101.Alarm);
(* notes on elements: Power Roller conv *)
(* Rung 9 *)
M03401_FB(Enable := P_On, RunFeedBack := XC0301_6_I[11], Tag := MO3401, ControlCom := A1_Control, OutputForward => XC0301_8_O[15], Alarm => MO3401.Alarm);
(* notes on elements: Labelling Conveyor motor *)
(* Rung 10 *)
MO2701_FB(Enable := P_On, RunFeedBack := XC0301_6_I[12], Tag := MO2701, ControlCom := A1_Control, OutputForward => XC0301_9_O[0], Alarm => MO2701.Alarm);
(* notes on elements: Top Tapping Machine Motor 1 *)
(* Rung 11 *)
MO2702_FB(Enable := P_On, RunFeedBack := XC0301_6_I[13], Tag := MO2702, ControlCom := A1_Control, OutputForward => XC0301_9_O[1], Alarm => MO2702.Alarm);
(* notes on elements: Top Tapping Machine Motor 2 *)

(* Section IDRob_SysOutputs: ladder, written here as Structured Text *)

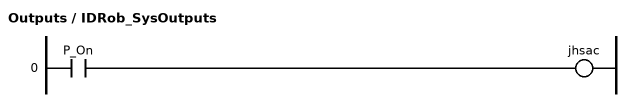
(* Rung 0 *)
jhsac := P_On;

(* Section IDRob_Outputs: ladder, written here as Structured Text *)

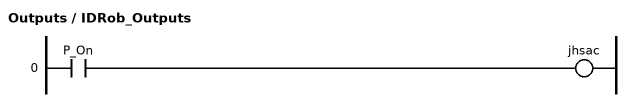
(* Rung 0 *)
jhsac := P_On;
END_PROGRAM

FUNCTION_BLOCK CYL
VAR
    ExSol : BOOL;
    RtSol : BOOL;
    CycleExtend : BOOL;
    CycleRetract : BOOL;
    TestCycleEnable : BOOL;
    CycleExtendtimer : TON;
    CycleRetracttimer : TON;
    ExtendTimer : TON;
    RetractTimer : TON;
    ExtendFaultTimer : TON;
    ExtendFault : BOOL;
    RetractFaultTimer : TON;
    RetractFault : BOOL;
    CycleExtendpre : TIME;
    CycleRetractpre : TIME;
    ExtendTime : TIME;
    RetractTime : TIME;
    ExtendTimeAcc : TIME;
    RetractTimeAcc : TIME;
    Timecal1 : LREAL;
    Timecal2 : LINT;
    Timecal3 : LREAL;
    Timecal4 : LINT;
    Timecal5 : LREAL;
    Timecal6 : LINT;
    Timecal7 : LREAL;
    Timecal8 : LINT;
    Timecal9 : LINT;
    Timecal10 : LREAL;
    Timecal11 : LINT;
    Timecal12 : LREAL;
END_VAR
VAR_INPUT
    Enable : BOOL;
END_VAR
VAR_OUTPUT
    EnableOut : BOOL;
    ExtendSol : BOOL;
    RetractSol : BOOL;
END_VAR
VAR_INPUT
    Extendreed1 : BOOL;
    Extendreed2 : BOOL;
    Retractreed1 : BOOL;
    Retractreed2 : BOOL;
    Accnowledge : BOOL;
END_VAR
VAR_IN_OUT
    Tag : CylinderD;
    ControlAlarm : BOOL;
END_VAR
VAR_OUTPUT
    Alarm : BOOL;
END_VAR
VAR
    _p1 : BOOL;
    _p2 : BOOL;
    _e3 : R_TRIG;
    _e4 : R_TRIG;
    _p5 : BOOL;
    _e6 : R_TRIG;
    _e7 : R_TRIG;
    _p8 : BOOL;
    _e9 : R_TRIG;
    _e10 : R_TRIG;
    _p11 : BOOL;
    _p12 : BOOL;
    _e13 : R_TRIG;
    _e14 : R_TRIG;
    _p15 : BOOL;
END_VAR
(* ladder, written here as Structured Text *)

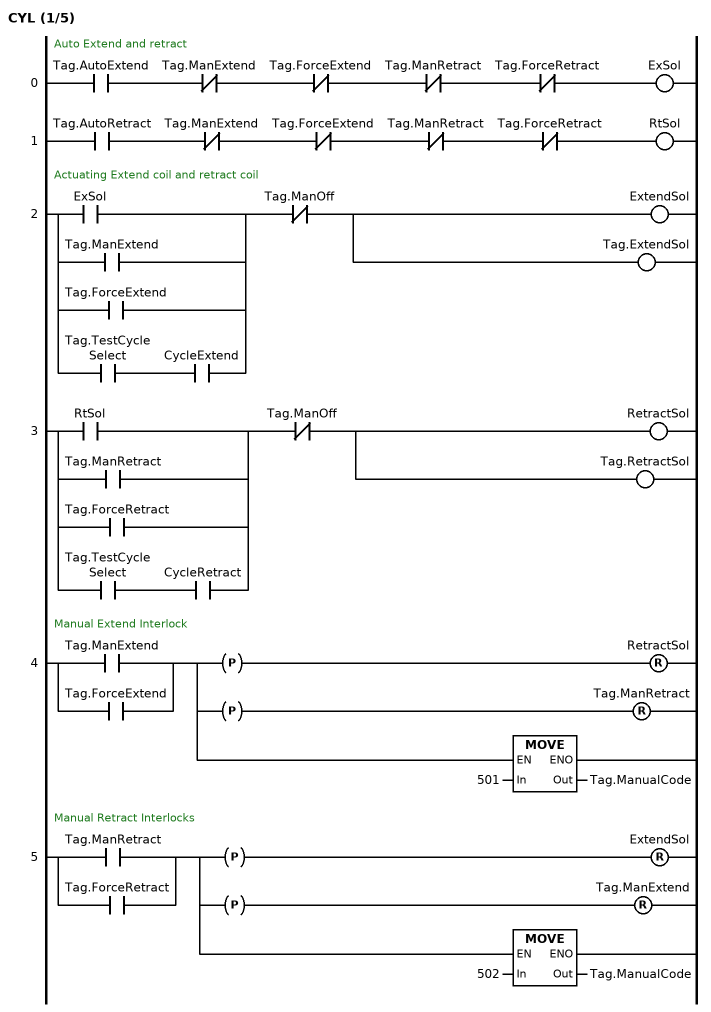
(* Rung 0: Auto Extend and retract *)
ExSol := Tag.AutoExtend AND NOT Tag.ManExtend AND NOT Tag.ForceExtend AND NOT Tag.ManRetract AND NOT Tag.ForceRetract;
(* Rung 1 *)
RtSol := Tag.AutoRetract AND NOT Tag.ManExtend AND NOT Tag.ForceExtend AND NOT Tag.ManRetract AND NOT Tag.ForceRetract;
(* Rung 2: Actuating Extend coil and retract coil *)
_p1 := (ExSol OR Tag.ManExtend OR Tag.ForceExtend OR (Tag.TestCycleSelect AND CycleExtend)) AND NOT Tag.ManOff;
ExtendSol := _p1;
Tag.ExtendSol := _p1;
(* Rung 3 *)
_p2 := (RtSol OR Tag.ManRetract OR Tag.ForceRetract OR (Tag.TestCycleSelect AND CycleRetract)) AND NOT Tag.ManOff;
RetractSol := _p2;
Tag.RetractSol := _p2;
(* Rung 4: Manual Extend Interlock *)
_e3(CLK := Tag.ManExtend OR Tag.ForceExtend);
IF _e3.Q THEN RetractSol := FALSE; END_IF;
_e4(CLK := Tag.ManExtend OR Tag.ForceExtend);
_p5 := Tag.ManExtend OR Tag.ForceExtend;
IF _e4.Q THEN Tag.ManRetract := FALSE; END_IF;
IF _p5 THEN Tag.ManualCode := 501; END_IF;
(* Rung 5: Manual Retract Interlocks *)
_e6(CLK := Tag.ManRetract OR Tag.ForceRetract);
IF _e6.Q THEN ExtendSol := FALSE; END_IF;
_e7(CLK := Tag.ManRetract OR Tag.ForceRetract);
_p8 := Tag.ManRetract OR Tag.ForceRetract;
IF _e7.Q THEN Tag.ManExtend := FALSE; END_IF;
IF _p8 THEN Tag.ManualCode := 502; END_IF;

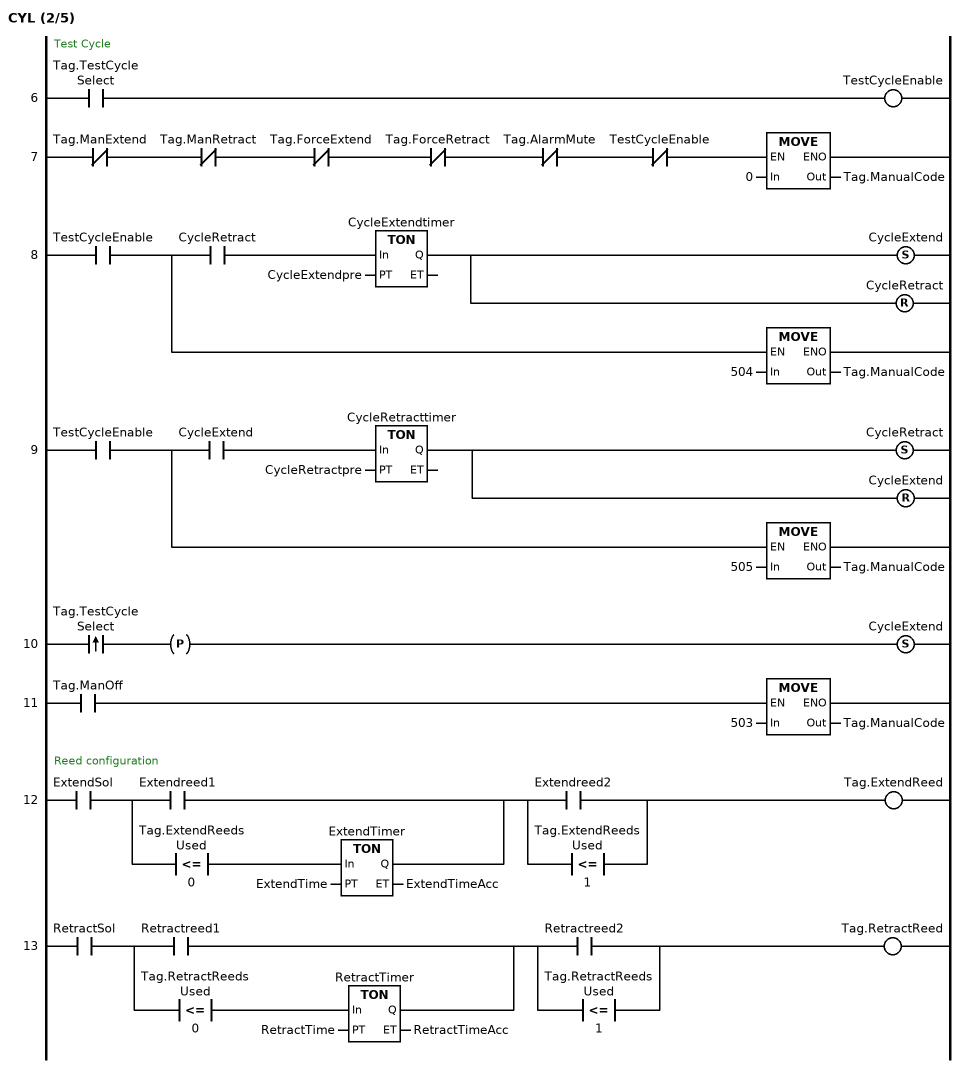
(* Rung 6: Test Cycle *)
TestCycleEnable := Tag.TestCycleSelect;
(* Rung 7 *)
IF NOT Tag.ManExtend AND NOT Tag.ManRetract AND NOT Tag.ForceExtend AND NOT Tag.ForceRetract AND NOT Tag.AlarmMute AND NOT TestCycleEnable THEN
    Tag.ManualCode := 0;
END_IF;
(* Rung 8 *)
CycleExtendtimer(In := TestCycleEnable AND CycleRetract, PT := CycleExtendpre);
IF CycleExtendtimer.Q THEN
    CycleExtend := TRUE;
    CycleRetract := FALSE;
END_IF;
IF TestCycleEnable THEN Tag.ManualCode := 504; END_IF;
(* Rung 9 *)
CycleRetracttimer(In := TestCycleEnable AND CycleExtend, PT := CycleRetractpre);
IF CycleRetracttimer.Q THEN
    CycleRetract := TRUE;
    CycleExtend := FALSE;
END_IF;
IF TestCycleEnable THEN Tag.ManualCode := 505; END_IF;
(* Rung 10 *)
_e9(CLK := Tag.TestCycleSelect);
_e10(CLK := _e9.Q);
IF _e10.Q THEN CycleExtend := TRUE; END_IF;
(* Rung 11 *)
IF Tag.ManOff THEN Tag.ManualCode := 503; END_IF;
(* Rung 12: Reed configuration *)
ExtendTimer(In := ExtendSol AND (Tag.ExtendReedsUsed <= 0), PT := ExtendTime, ET => ExtendTimeAcc);
Tag.ExtendReed := ((ExtendSol AND Extendreed1) OR ExtendTimer.Q) AND (Extendreed2 OR (Tag.ExtendReedsUsed <= 1));
(* Rung 13 *)
RetractTimer(In := RetractSol AND (Tag.RetractReedsUsed <= 0), PT := RetractTime, ET => RetractTimeAcc);
Tag.RetractReed := ((RetractSol AND Retractreed1) OR RetractTimer.Q) AND (Retractreed2 OR (Tag.RetractReedsUsed <= 1));

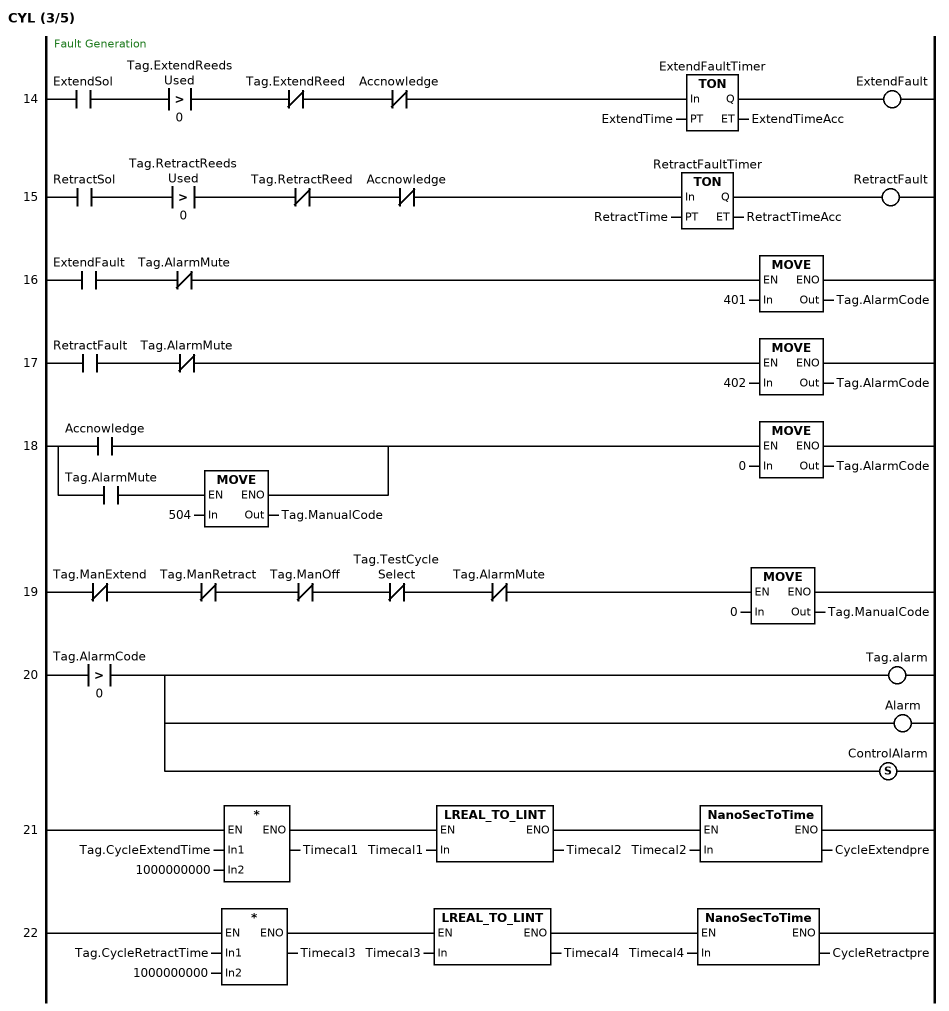
(* Rung 14: Fault Generation *)
ExtendFaultTimer(In := ExtendSol AND (Tag.ExtendReedsUsed > 0) AND NOT Tag.ExtendReed AND NOT Accnowledge, PT := ExtendTime, ET => ExtendTimeAcc);
ExtendFault := ExtendFaultTimer.Q;
(* Rung 15 *)
RetractFaultTimer(In := RetractSol AND (Tag.RetractReedsUsed > 0) AND NOT Tag.RetractReed AND NOT Accnowledge, PT := RetractTime, ET => RetractTimeAcc);
RetractFault := RetractFaultTimer.Q;
(* Rung 16 *)
IF ExtendFault AND NOT Tag.AlarmMute THEN Tag.AlarmCode := 401; END_IF;
(* Rung 17 *)
IF RetractFault AND NOT Tag.AlarmMute THEN Tag.AlarmCode := 402; END_IF;
(* Rung 18 *)
_p11 := Tag.AlarmMute;
IF _p11 THEN Tag.ManualCode := 504; END_IF;
IF Accnowledge OR _p11 THEN Tag.AlarmCode := 0; END_IF;
(* Rung 19 *)
IF NOT Tag.ManExtend AND NOT Tag.ManRetract AND NOT Tag.ManOff AND NOT Tag.TestCycleSelect AND NOT Tag.AlarmMute THEN
    Tag.ManualCode := 0;
END_IF;
(* Rung 20 *)
_p12 := Tag.AlarmCode > 0;
Tag.alarm := _p12;
Alarm := _p12;
IF _p12 THEN ControlAlarm := TRUE; END_IF;
(* Rung 21 *)
Timecal1 := Tag.CycleExtendTime * 1000000000;
Timecal2 := LREAL_TO_LINT(In := Timecal1);
CycleExtendpre := NanoSecToTime(In := Timecal2);
(* Rung 22 *)
Timecal3 := Tag.CycleRetractTime * 1000000000;
Timecal4 := LREAL_TO_LINT(In := Timecal3);
CycleRetractpre := NanoSecToTime(In := Timecal4);

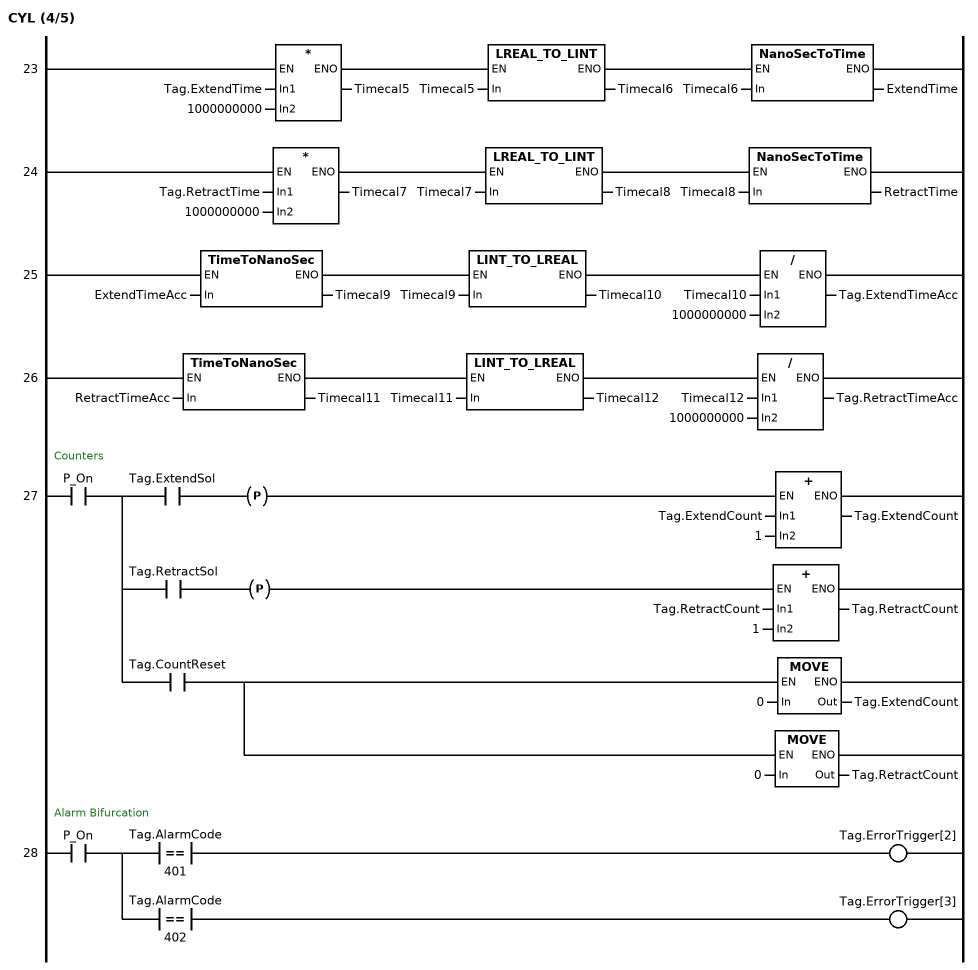
(* Rung 23 *)
Timecal5 := Tag.ExtendTime * 1000000000;
Timecal6 := LREAL_TO_LINT(In := Timecal5);
ExtendTime := NanoSecToTime(In := Timecal6);
(* Rung 24 *)
Timecal7 := Tag.RetractTime * 1000000000;
Timecal8 := LREAL_TO_LINT(In := Timecal7);
RetractTime := NanoSecToTime(In := Timecal8);
(* Rung 25 *)
Timecal9 := TimeToNanoSec(In := ExtendTimeAcc);
Timecal10 := LINT_TO_LREAL(In := Timecal9);
Tag.ExtendTimeAcc := Timecal10 / 1000000000;
(* Rung 26 *)
Timecal11 := TimeToNanoSec(In := RetractTimeAcc);
Timecal12 := LINT_TO_LREAL(In := Timecal11);
Tag.RetractTimeAcc := Timecal12 / 1000000000;
(* Rung 27: Counters *)
_e13(CLK := P_On AND Tag.ExtendSol);
IF _e13.Q THEN Tag.ExtendCount := Tag.ExtendCount + 1; END_IF;
_e14(CLK := P_On AND Tag.RetractSol);
IF _e14.Q THEN Tag.RetractCount := Tag.RetractCount + 1; END_IF;
_p15 := P_On AND Tag.CountReset;
IF _p15 THEN
    Tag.ExtendCount := 0;
    Tag.RetractCount := 0;
END_IF;
(* Rung 28: Alarm Bifurcation *)
Tag.ErrorTrigger[2] := P_On AND (Tag.AlarmCode = 401);
Tag.ErrorTrigger[3] := P_On AND (Tag.AlarmCode = 402);

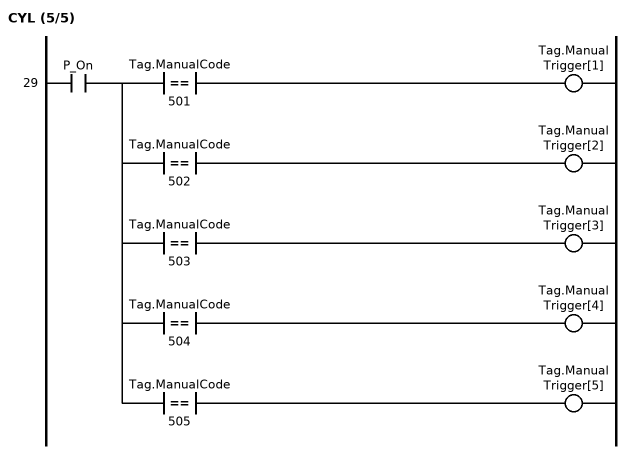
(* Rung 29 *)
Tag.ManualTrigger[1] := P_On AND (Tag.ManualCode = 501);
Tag.ManualTrigger[2] := P_On AND (Tag.ManualCode = 502);
Tag.ManualTrigger[3] := P_On AND (Tag.ManualCode = 503);
Tag.ManualTrigger[4] := P_On AND (Tag.ManualCode = 504);
Tag.ManualTrigger[5] := P_On AND (Tag.ManualCode = 505);
END_FUNCTION_BLOCK

FUNCTION_BLOCK Servo
VAR
    MCPower : MC_Power;
    MCHome : MC_Home;
    MCJOG : MC_MoveJog;
    MCManualmov : MC_MoveJog;
    MCManualJog : MC_MoveAbsolute;
    MCMovePos1 : MC_MoveAbsolute;
    MCMovePos2 : MC_MoveAbsolute;
    MCMovePos3 : MC_MoveAbsolute;
    MCMovePos4 : MC_MoveAbsolute;
END_VAR
VAR RETAIN
    Pos1Speed : LREAL;
    Pos1Acceleration : LREAL;
    Pos1Deceleration : LREAL;
    Pos1Jerk : LREAL;
END_VAR
VAR
    Pos2Speed : LREAL;
    Pos2Acceleration : LREAL;
    Pos2Deceleration : LREAL;
    Pos2Jerk : LREAL;
    Pos3Speed : LREAL;
    Pos3Acceleration : LREAL;
    Pos3Deceleration : LREAL;
    Pos3Jerk : LREAL;
    Pos4Speed : LREAL;
    Pos4Acceleration : LREAL;
    Pos4Deceleration : LREAL;
    Pos4Jerk : LREAL;
    Pos4MoveType : _eMC_DIRECTION;
    Pos2MoveType : _eMC_DIRECTION;
    Pos3MoveType : _eMC_DIRECTION;
END_VAR
VAR RETAIN
    Pos1MoveType : _eMC_DIRECTION;
END_VAR
VAR
    MC_Movezero : MC_MoveZeroPosition;
    SpeedCal1 : LREAL;
END_VAR
VAR RETAIN
    Jerk : LREAL;
END_VAR
VAR
    Updated : BOOL;
    MCMoveVel : MC_MoveVelocity;
    Pos1PosTol : LREAL;
    Pos1NegTol : LREAL;
    Pos2PosTol : LREAL;
    Pos2NegTol : LREAL;
    Pos3PosTol : LREAL;
    Pos3NegTol : LREAL;
    Pos4PosTol : LREAL;
    Pos4NegTol : LREAL;
END_VAR
VAR RETAIN
    Temp : DWORD;
END_VAR
VAR
    JogType : _eMC_DIRECTION;
    MoveVeltype : _eMC_DIRECTION;
    Runhourstimer : TON;
    RunHoursT : TIME;
    RunHours : ARRAY[0..1] OF LINT;
    RunHour : REAL;
    Alarmmonitor : ATC_E\oneS\oneS_Monitor;
    Monitors : ATC_E\oneS\sOneSData;
    Time_out_data : UINT;
    DeviceData : ATC_E\oneS\sDeviceData;
    zcom : BOOL;
    zcom6 : BOOL;
    MCMovePos5 : MC_MoveAbsolute;
    Pos5MoveType : _eMC_DIRECTION;
    Pos5PosTol : LREAL;
    Pos5NegTol : LREAL;
    MCMovePos6 : MC_MoveAbsolute;
    Pos6MoveType : _eMC_DIRECTION;
    Pos6PosTol : LREAL;
    Pos6NegTol : LREAL;
END_VAR
VAR_INPUT
    Enable : BOOL;
END_VAR
VAR_OUTPUT
    EnableOut : BOOL;
END_VAR
VAR_IN_OUT CONSTANT
    Axis : _sAXIS_REF;
END_VAR
VAR_IN_OUT
    Tag : ServoD;
END_VAR
VAR_OUTPUT
    Alarm : BOOL;
END_VAR
VAR_IN_OUT
    ControlAlarm : BOOL;
END_VAR
VAR
    _p1 : BOOL;
    _e2 : R_TRIG;
END_VAR
(* ladder, written here as Structured Text *)

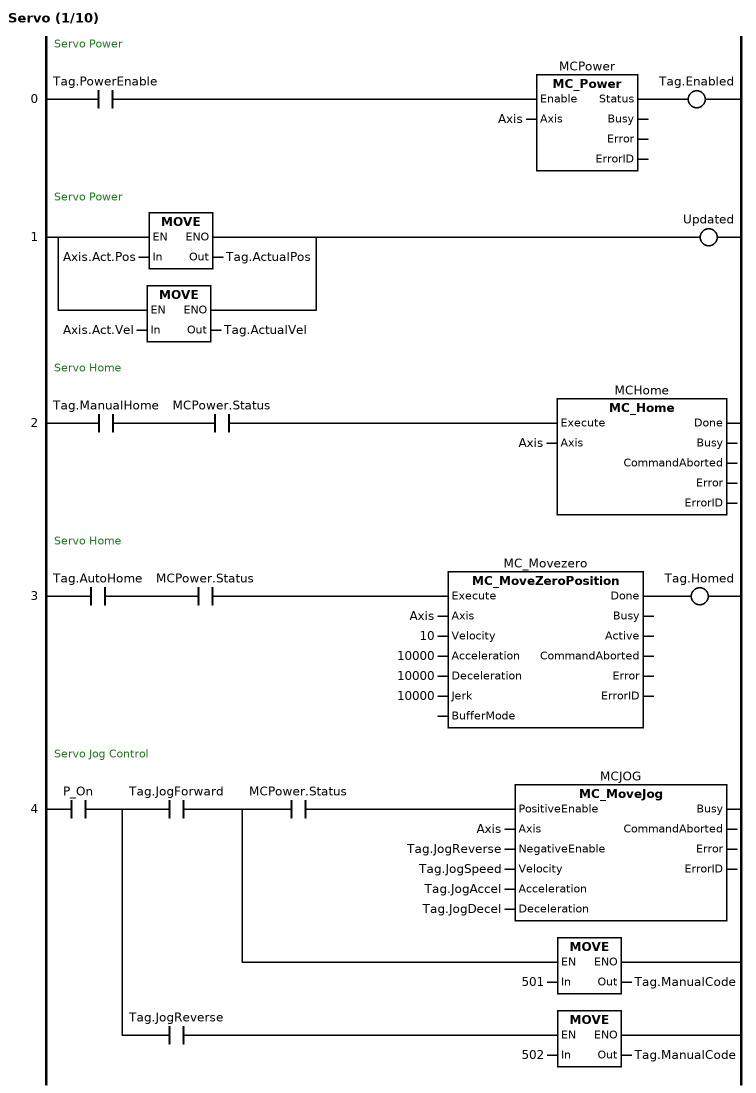
(* Rung 0: Servo Power *)
MCPower(Enable := Tag.PowerEnable, Axis := Axis);
Tag.Enabled := MCPower.Status;
(* Rung 1: Servo Power *)
Tag.ActualPos := Axis.Act.Pos;
Tag.ActualVel := Axis.Act.Vel;
Updated := TRUE;
(* Rung 2: Servo Home *)
MCHome(Execute := Tag.ManualHome AND MCPower.Status, Axis := Axis);
(* Rung 3: Servo Home *)
MC_Movezero(Execute := Tag.AutoHome AND MCPower.Status, Axis := Axis, Velocity := 10, Acceleration := 10000, Deceleration := 10000, Jerk := 10000);
Tag.Homed := MC_Movezero.Done;
(* Rung 4: Servo Jog Control *)
MCJOG(PositiveEnable := P_On AND Tag.JogForward AND MCPower.Status, Axis := Axis, NegativeEnable := Tag.JogReverse, Velocity := Tag.JogSpeed, Acceleration := Tag.JogAccel, Deceleration := Tag.JogDecel);
IF P_On AND Tag.JogForward THEN Tag.ManualCode := 501; END_IF;
IF P_On AND Tag.JogReverse THEN Tag.ManualCode := 502; END_IF;

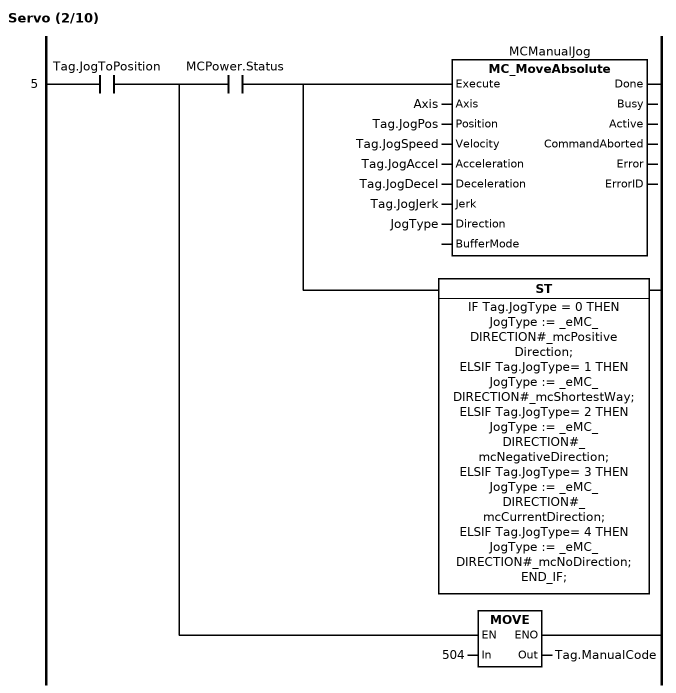
(* Rung 5 *)
MCManualJog(Execute := Tag.JogToPosition AND MCPower.Status, Axis := Axis, Position := Tag.JogPos, Velocity := Tag.JogSpeed, Acceleration := Tag.JogAccel, Deceleration := Tag.JogDecel, Jerk := Tag.JogJerk, Direction := JogType);
IF Tag.JogToPosition AND MCPower.Status THEN
    IF Tag.JogType = 0 THEN
    JogType := _eMC_DIRECTION#_mcPositiveDirection;
    ELSIF Tag.JogType= 1 THEN
    JogType := _eMC_DIRECTION#_mcShortestWay;
    ELSIF Tag.JogType= 2 THEN
    JogType := _eMC_DIRECTION#_mcNegativeDirection;
    ELSIF Tag.JogType= 3 THEN
    JogType := _eMC_DIRECTION#_mcCurrentDirection;
    ELSIF Tag.JogType= 4 THEN
    JogType := _eMC_DIRECTION#_mcNoDirection;
    END_IF;
END_IF;
IF Tag.JogToPosition THEN Tag.ManualCode := 504; END_IF;

